(* IEC 61131-3 sources: MSMP/PLC_Master/Source/Global, 2 files *)

(* ---- G_RuntimeDB.st ---- *)
VAR_GLOBAL
 gRuntimeDB : ST_RuntimeDB;
END_VAR

(* ---- G_Stations.st ---- *)
VAR_GLOBAL
    Stations : ARRAY[1..11] OF ST_Station;
END_VAR
